// TIA Portal V20 export
FUNCTION_BLOCK "FB_Pos16"   // FB30141, LAD
{ S7_Optimized_Access := 'TRUE' }
// stored: AutoNumber false, MemoryReserve 100, SetENOAutomatically false
   VAR_INPUT
      Opmode { ExternalAccessible := 'False'; ExternalVisible := 'False'; ExternalWritable := 'False'} : "OPMODE_OUT_UDT";
      TO_PosAxis : TO_PositioningAxis;
      I_iNum_Abspos : Int;
      I_bMan_Enable : Bool;
   END_VAR
   VAR_IN_OUT
      Ds_Pos16 : "sPos16";
   END_VAR
   VAR
      instAxis01 { ExternalAccessible := 'False'; ExternalVisible := 'False'; ExternalWritable := 'False'} : "LAxisCtrl_PosAxis";
      instShearAxisStatus { S7_SetPoint := 'True'} : "LAxisCtrl_GetAxisStatusWord";
      RT_Reset { S7_SetPoint := 'True'} : R_TRIG;
      RT_PB { ExternalAccessible := 'False'; ExternalVisible := 'False'; ExternalWritable := 'False'} : Array[0..19] of R_TRIG;   // Störungen / Alarms
      FT_PB { ExternalAccessible := 'False'; ExternalVisible := 'False'; ExternalWritable := 'False'; S7_SetPoint := 'True'} : Array[0..19] of F_TRIG;   // Störungen unterdrücken, Belegung identisch mit "Alarm" / Hide Alarms, identical with "Alarm"
      TON_PB { ExternalAccessible := 'False'; ExternalVisible := 'False'; ExternalWritable := 'False'} : Array[0..19] of TON_TIME;   // Fallende Flanke / Falling edge
      TOF_PB { ExternalAccessible := 'False'; ExternalVisible := 'False'; ExternalWritable := 'False'} : Array[0..19] of TOF_TIME;   // Negativer Impuls / Negative pulse
      i { S7_SetPoint := 'True'} : Int;
      temp_cmd_bEnableAxis { ExternalAccessible := 'False'; ExternalVisible := 'False'; ExternalWritable := 'False'} : Bool;
      temp_cmd_bresetAxis { ExternalAccessible := 'False'; ExternalVisible := 'False'; ExternalWritable := 'False'} : Bool;
      temp_cmd_bjogForward { ExternalAccessible := 'False'; ExternalVisible := 'False'; ExternalWritable := 'False'} : Bool;
      temp_cmd_bjogBackward { ExternalAccessible := 'False'; ExternalVisible := 'False'; ExternalWritable := 'False'} : Bool;
      temp_cmd_bmoveVelocity { ExternalAccessible := 'False'; ExternalVisible := 'False'; ExternalWritable := 'False'} : Bool;
      temp_cmd_bstop { ExternalAccessible := 'False'; ExternalVisible := 'False'; ExternalWritable := 'False'} : Bool;
      temp_cmd_bfastStop { ExternalAccessible := 'False'; ExternalVisible := 'False'; ExternalWritable := 'False'} : Bool;
      temp_cmd_bhoming { ExternalAccessible := 'False'; ExternalVisible := 'False'; ExternalWritable := 'False'} : Bool;
      temp_cmd_bGoToPos { ExternalAccessible := 'False'; ExternalVisible := 'False'; ExternalWritable := 'False'} : Array[0..16] of Bool;
      temp_cmd_iGoToPos : Word;
      temp_cmd_bCallAbsPos : Bool;
      temp_cmd_bRelPos : Bool;
      temp_Para_rJog_Speed { ExternalAccessible := 'False'; ExternalVisible := 'False'; ExternalWritable := 'False'} : LReal;
      temp_configuration { ExternalAccessible := 'False'; ExternalVisible := 'False'; ExternalWritable := 'False'} : "LAxisCtrl_typeAxisConfig";   // Diagnostics structure
      temp_Status { ExternalAccessible := 'False'; ExternalVisible := 'False'; ExternalWritable := 'False'} : Word;
      temp_AxisEnabled { ExternalAccessible := 'False'; ExternalVisible := 'False'; ExternalWritable := 'False'} : Bool;
      temp_CommandBusy { ExternalAccessible := 'False'; ExternalVisible := 'False'; ExternalWritable := 'False'} : Bool;
      temp_CommandDone { ExternalAccessible := 'False'; ExternalVisible := 'False'; ExternalWritable := 'False'} : Bool;
      temp_CommandAborted { ExternalAccessible := 'False'; ExternalVisible := 'False'; ExternalWritable := 'False'} : Bool;
      temp_InVelocity { ExternalAccessible := 'False'; ExternalVisible := 'False'; ExternalWritable := 'False'} : Bool;
      temp_jogSelected { ExternalAccessible := 'False'; ExternalVisible := 'False'; ExternalWritable := 'False'} : Bool;
      tempPosAbsoluteSelected { ExternalAccessible := 'False'; ExternalVisible := 'False'; ExternalWritable := 'False'} : Bool;
      temp_diagnostics { ExternalAccessible := 'False'; ExternalVisible := 'False'; ExternalWritable := 'False'} : "LAxisCtrl_typeDiagnostics";
      temp_stop_Dec { ExternalAccessible := 'False'; ExternalVisible := 'False'; ExternalWritable := 'False'} : LReal;
      temp_faststop_Dec { ExternalAccessible := 'False'; ExternalVisible := 'False'; ExternalWritable := 'False'} : LReal;
      temp_cmd_bGoToPosAll : Bool;
      temp_iFBStatus : Word;
      temp_iMCStatus : Word;
      old_iFBStatus : Word;
      old_iMCStatus : Word;
   END_VAR
BEGIN

REGION Network 1
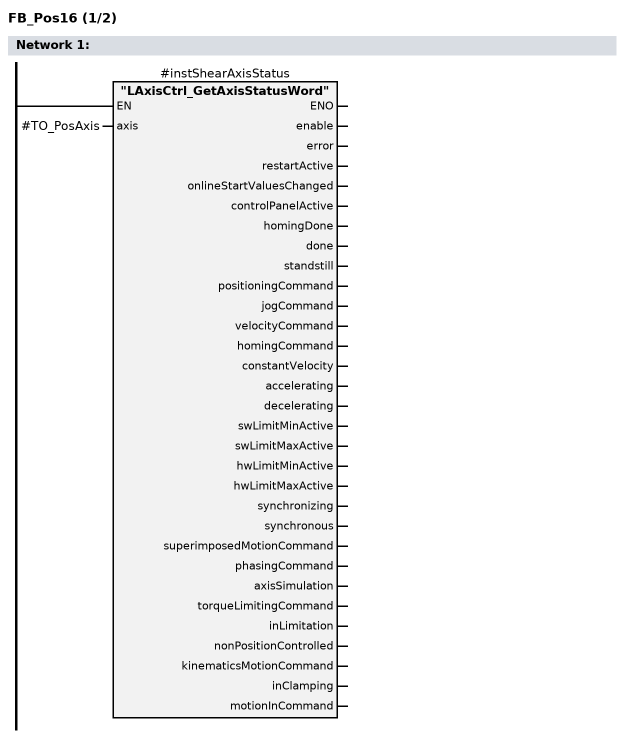
   RUNG wire#powerrail
      #instShearAxisStatus(axis := #TO_PosAxis, enable =>, error =>, restartActive =>, onlineStartValuesChanged =>, controlPanelActive =>, homingDone =>, done =>, standstill =>, positioningCommand =>, jogCommand =>, velocityCommand =>, homingCommand =>, constantVelocity =>, accelerating =>, decelerating =>, swLimitMinActive =>, swLimitMaxActive =>, hwLimitMinActive =>, hwLimitMaxActive =>, synchronizing =>, synchronous =>, superimposedMotionCommand =>, phasingCommand =>, axisSimulation =>, torqueLimitingCommand =>, inLimitation =>, nonPositionControlled =>, kinematicsMotionCommand =>, inClamping =>, motionInCommand =>)
   END_RUNG
   // the same network as SCL:
   #instShearAxisStatus(axis := #TO_PosAxis);   // "LAxisCtrl_GetAxisStatusWord"
END_REGION

REGION Network 2: LAxisCtrl
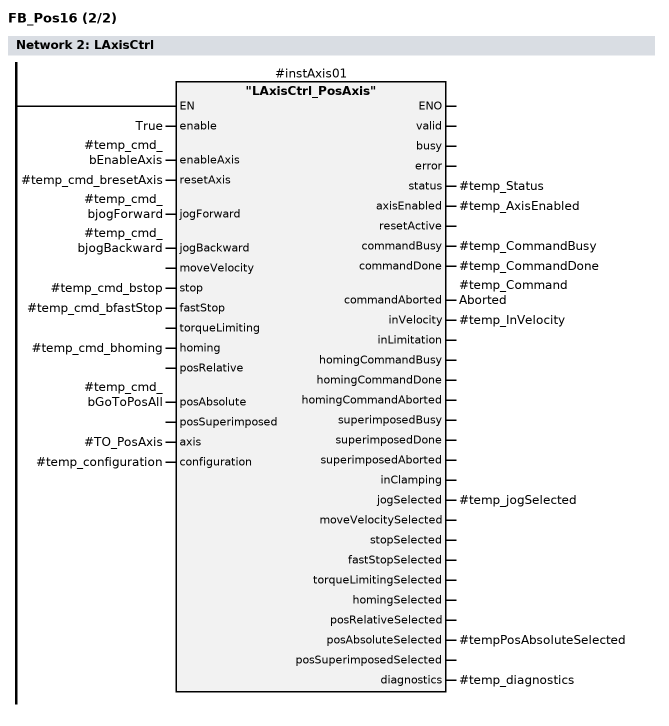
   RUNG wire#powerrail
      #instAxis01(enable := True, enableAxis := #temp_cmd_bEnableAxis, resetAxis := #temp_cmd_bresetAxis, jogForward := #temp_cmd_bjogForward, jogBackward := #temp_cmd_bjogBackward, moveVelocity :=, stop := #temp_cmd_bstop, fastStop := #temp_cmd_bfastStop, torqueLimiting :=, homing := #temp_cmd_bhoming, posRelative :=, posAbsolute := #temp_cmd_bGoToPosAll, posSuperimposed :=, axis := #TO_PosAxis, configuration := #temp_configuration, valid =>, busy =>, error =>, status => #temp_Status, axisEnabled => #temp_AxisEnabled, resetActive =>, commandBusy => #temp_CommandBusy, commandDone => #temp_CommandDone, commandAborted => #temp_CommandAborted, inVelocity => #temp_InVelocity, inLimitation =>, homingCommandBusy =>, homingCommandDone =>, homingCommandAborted =>, superimposedBusy =>, superimposedDone =>, superimposedAborted =>, inClamping =>, jogSelected => #temp_jogSelected, moveVelocitySelected =>, stopSelected =>, fastStopSelected =>, torqueLimitingSelected =>, homingSelected =>, posRelativeSelected =>, posAbsoluteSelected => #tempPosAbsoluteSelected, posSuperimposedSelected =>, diagnostics => #temp_diagnostics)
   END_RUNG
   // the same network as SCL:
   #instAxis01(enable := True,   // "LAxisCtrl_PosAxis"
               enableAxis := #temp_cmd_bEnableAxis,
               resetAxis := #temp_cmd_bresetAxis,
               jogForward := #temp_cmd_bjogForward,
               jogBackward := #temp_cmd_bjogBackward,
               stop := #temp_cmd_bstop,
               fastStop := #temp_cmd_bfastStop,
               homing := #temp_cmd_bhoming,
               posAbsolute := #temp_cmd_bGoToPosAll,
               axis := #TO_PosAxis,
               configuration := #temp_configuration,
               status => #temp_Status,
               axisEnabled => #temp_AxisEnabled,
               commandBusy => #temp_CommandBusy,
               commandDone => #temp_CommandDone,
               commandAborted => #temp_CommandAborted,
               inVelocity => #temp_InVelocity,
               jogSelected => #temp_jogSelected,
               posAbsoluteSelected => #tempPosAbsoluteSelected,
               diagnostics => #temp_diagnostics);
END_REGION

REGION Network 3 (SCL): input
   #temp_cmd_bEnableAxis  := #Ds_Pos16.I_CMD_bEnableAxis OR (#Ds_Pos16.I_HMI_bEnableAxis AND #I_bMan_Enable);
   #temp_cmd_bresetAxis   := #Ds_Pos16.I_CMD_bResetAxis;
   #temp_cmd_bjogForward  := #Ds_Pos16.I_InLock_bjogForward AND (#Ds_Pos16.I_CMD_bjogForward OR (#Ds_Pos16.I_HMI_bjogForward AND #I_bMan_Enable));
   #temp_cmd_bjogBackward := #Ds_Pos16.I_InLock_bjogBackward AND (#Ds_Pos16.I_CMD_bjogBackward OR (#Ds_Pos16.I_HMI_bjogBackward AND #I_bMan_Enable));
   #temp_cmd_bstop        := #Ds_Pos16.I_CMD_bstop OR (#Ds_Pos16.I_HMI_bstop AND #I_bMan_Enable);
   #temp_cmd_bfastStop    := #Ds_Pos16.I_CMD_bfastStop;
   #temp_cmd_bhoming      := #Ds_Pos16.I_InLock_bHoming AND (#Ds_Pos16.I_CMD_bHoming OR #Ds_Pos16.I_HMI_bHoming);
END_REGION

REGION Network 4 (SCL): Configuration
   #Ds_Pos16.I_Para_rJog_Speed[0] := 10.0;
   #Ds_Pos16.I_Para_rMV_Speed[0]  := 10.0;
   #Ds_Pos16.I_Para_rStop_Dec[0]  := 20.0;
   #Ds_Pos16.I_Para_rEStop_Dec[0] := 50.0;

   #Ds_Pos16.I_Para_rJog_Speed[1] := 10.0 * #Ds_Pos16.I_Para_rJog_Speed[0];
   #Ds_Pos16.I_Para_rJog_Speed[2] := 10.0 * #Ds_Pos16.I_Para_rJog_Speed[0];
   #Ds_Pos16.I_Para_rMV_Speed[1] := 10.0 * #Ds_Pos16.I_Para_rMV_Speed[0];
   #Ds_Pos16.I_Para_rMV_Speed[2] := 10.0 * #Ds_Pos16.I_Para_rMV_Speed[0];
   #Ds_Pos16.I_Para_rStop_Dec[1] := 100.0 * #Ds_Pos16.I_Para_rStop_Dec[0];
   #Ds_Pos16.I_Para_rEStop_Dec[1] := 100.0 * #Ds_Pos16.I_Para_rEStop_Dec[0];

   IF #temp_configuration.jog.velocity <> #Ds_Pos16.I_Para_rJog_Speed[0] OR
       #temp_configuration.jog.acceleration <> #Ds_Pos16.I_Para_rJog_Speed[1] OR
       #temp_configuration.jog.deceleration <> #Ds_Pos16.I_Para_rJog_Speed[2] OR
       #temp_configuration.moveVelocity.acceleration <> #Ds_Pos16.I_Para_rMV_Speed[0] OR
       #temp_configuration.moveVelocity.deceleration <> #Ds_Pos16.I_Para_rMV_Speed[1] OR
       #temp_configuration.moveVelocity.acceleration <> #Ds_Pos16.I_Para_rMV_Speed[2] OR
       #temp_configuration.stop.deceleration <> #Ds_Pos16.I_Para_rStop_Dec[0] OR
       #temp_configuration.stop.jerk <> #Ds_Pos16.I_Para_rStop_Dec[1] OR
       #temp_configuration.fastStop.deceleration <> #Ds_Pos16.I_Para_rEStop_Dec[0] OR
       #temp_configuration.fastStop.jerk <> #Ds_Pos16.I_Para_rEStop_Dec[1]
   THEN
       // Jog
       #temp_configuration.jog.velocity := #Ds_Pos16.I_Para_rJog_Speed[0];
       #temp_configuration.jog.acceleration := #Ds_Pos16.I_Para_rJog_Speed[1];
       #temp_configuration.jog.deceleration := #Ds_Pos16.I_Para_rJog_Speed[2];
       // Move
       #temp_configuration.moveVelocity.velocity := #Ds_Pos16.I_Para_rMV_Speed[0];
       #temp_configuration.moveVelocity.acceleration := #Ds_Pos16.I_Para_rMV_Speed[1];
       #temp_configuration.moveVelocity.deceleration := #Ds_Pos16.I_Para_rMV_Speed[2];
       // Stop   
       #temp_configuration.stop.deceleration := #Ds_Pos16.I_Para_rStop_Dec[0];
       #temp_configuration.stop.jerk := #Ds_Pos16.I_Para_rStop_Dec[1];
       //faststoo
       #temp_configuration.fastStop.deceleration := #Ds_Pos16.I_Para_rEStop_Dec[0];
       #temp_configuration.fastStop.jerk := #Ds_Pos16.I_Para_rEStop_Dec[1];
   END_IF;

   // Homing
   #temp_configuration.homing.mode := 0;//I_iHomeMode
   #temp_configuration.homing.position := 0;//I_iHomePos

   //abspos
   FOR #i := 1 TO 16 DO
       #Ds_Pos16.I_Para_rAcc_Set[#i] := 10.0 * #Ds_Pos16.I_Para_rSpeed_Abs[0];
       #Ds_Pos16.I_Para_rDec_Set[#i] := 10.0 * #Ds_Pos16.I_Para_rSpeed_Abs[0];
       #Ds_Pos16.I_Para_rJerk_Set[#i] := 100.0 * #Ds_Pos16.I_Para_rSpeed_Abs[0];
   END_FOR;


   //#temp_posAbsolute := (#Ds_Pos16.I_CMD_iGoToPos <> 16#0);
   #temp_cmd_bGoToPos[1] := ((#Opmode.Automatic_active=1 AND #Ds_Pos16.I_CMD_iGoToPos = 1) OR (#Opmode.Manual_active AND #Ds_Pos16.I_HMI_iGoToPos = 1)) AND #Ds_Pos16.I_InLock_bGoToPos[1];
   #temp_cmd_bGoToPos[2] := ((#Opmode.Automatic_active=1 AND #Ds_Pos16.I_CMD_iGoToPos = 2) OR (#Opmode.Manual_active AND  #Ds_Pos16.I_HMI_iGoToPos = 2)) AND #Ds_Pos16.I_InLock_bGoToPos[2];
   #temp_cmd_bGoToPos[3] := ((#Opmode.Automatic_active=1 AND #Ds_Pos16.I_CMD_iGoToPos = 3) OR (#Opmode.Manual_active AND  #Ds_Pos16.I_HMI_iGoToPos = 3)) AND #Ds_Pos16.I_InLock_bGoToPos[3];
   #temp_cmd_bGoToPos[4] := ((#Opmode.Automatic_active=1 AND #Ds_Pos16.I_CMD_iGoToPos = 4) OR (#Opmode.Manual_active AND  #Ds_Pos16.I_HMI_iGoToPos = 4)) AND #Ds_Pos16.I_InLock_bGoToPos[4];
   #temp_cmd_bGoToPos[5] := ((#Opmode.Automatic_active=1 AND #Ds_Pos16.I_CMD_iGoToPos = 5) OR (#Opmode.Manual_active AND  #Ds_Pos16.I_HMI_iGoToPos = 5)) AND #Ds_Pos16.I_InLock_bGoToPos[5];
   #temp_cmd_bGoToPos[6] := ((#Opmode.Automatic_active=1 AND #Ds_Pos16.I_CMD_iGoToPos = 6) OR (#Opmode.Manual_active AND  #Ds_Pos16.I_HMI_iGoToPos = 6)) AND #Ds_Pos16.I_InLock_bGoToPos[6];
   #temp_cmd_bGoToPos[7] := ((#Opmode.Automatic_active=1 AND #Ds_Pos16.I_CMD_iGoToPos = 7) OR (#Opmode.Manual_active AND  #Ds_Pos16.I_HMI_iGoToPos = 7)) AND #Ds_Pos16.I_InLock_bGoToPos[7];
   #temp_cmd_bGoToPos[8] := ((#Opmode.Automatic_active=1 AND #Ds_Pos16.I_CMD_iGoToPos = 8) OR (#Opmode.Manual_active AND  #Ds_Pos16.I_HMI_iGoToPos = 8)) AND #Ds_Pos16.I_InLock_bGoToPos[8];
   #temp_cmd_bGoToPos[9] := ((#Opmode.Automatic_active=1 AND #Ds_Pos16.I_CMD_iGoToPos = 9) OR (#Opmode.Manual_active AND  #Ds_Pos16.I_HMI_iGoToPos = 9)) AND #Ds_Pos16.I_InLock_bGoToPos[9];
   #temp_cmd_bGoToPos[10] := ((#Opmode.Automatic_active=1 AND #Ds_Pos16.I_CMD_iGoToPos = 10) OR (#Opmode.Manual_active AND  #Ds_Pos16.I_HMI_iGoToPos = 10)) AND #Ds_Pos16.I_InLock_bGoToPos[10];
   #temp_cmd_bGoToPos[11] := ((#Opmode.Automatic_active=1 AND #Ds_Pos16.I_CMD_iGoToPos = 11) OR (#Opmode.Manual_active AND  #Ds_Pos16.I_HMI_iGoToPos = 11)) AND #Ds_Pos16.I_InLock_bGoToPos[11];
   #temp_cmd_bGoToPos[12] := ((#Opmode.Automatic_active=1 AND #Ds_Pos16.I_CMD_iGoToPos = 12) OR (#Opmode.Manual_active AND  #Ds_Pos16.I_HMI_iGoToPos = 12)) AND #Ds_Pos16.I_InLock_bGoToPos[12];
   #temp_cmd_bGoToPos[13] := ((#Opmode.Automatic_active=1 AND #Ds_Pos16.I_CMD_iGoToPos = 13) OR (#Opmode.Manual_active AND  #Ds_Pos16.I_HMI_iGoToPos = 13)) AND #Ds_Pos16.I_InLock_bGoToPos[13];
   #temp_cmd_bGoToPos[14] := ((#Opmode.Automatic_active=1 AND #Ds_Pos16.I_CMD_iGoToPos = 14) OR (#Opmode.Manual_active AND  #Ds_Pos16.I_HMI_iGoToPos = 14)) AND #Ds_Pos16.I_InLock_bGoToPos[14];
   #temp_cmd_bGoToPos[15] := ((#Opmode.Automatic_active=1 AND #Ds_Pos16.I_CMD_iGoToPos = 15) OR (#Opmode.Manual_active AND  #Ds_Pos16.I_HMI_iGoToPos = 15)) AND #Ds_Pos16.I_InLock_bGoToPos[15];
   #temp_cmd_bGoToPos[16] := ((#Opmode.Automatic_active=1 AND #Ds_Pos16.I_CMD_iGoToPos = 16) OR (#Opmode.Manual_active AND  #Ds_Pos16.I_HMI_iGoToPos = 16)) AND #Ds_Pos16.I_InLock_bGoToPos[16];

   #temp_cmd_bGoToPosAll := #temp_cmd_bGoToPos[1] OR #temp_cmd_bGoToPos[2] OR #temp_cmd_bGoToPos[3] OR #temp_cmd_bGoToPos[4]
   OR #temp_cmd_bGoToPos[5] OR #temp_cmd_bGoToPos[6] OR #temp_cmd_bGoToPos[7] OR #temp_cmd_bGoToPos[8]
   OR #temp_cmd_bGoToPos[9] OR #temp_cmd_bGoToPos[10] OR #temp_cmd_bGoToPos[11] OR #temp_cmd_bGoToPos[12]
   OR #temp_cmd_bGoToPos[13] OR #temp_cmd_bGoToPos[14] OR #temp_cmd_bGoToPos[15] OR #temp_cmd_bGoToPos[16]
   ;
   //#temp_posAbsolute :=
   //#Ds_Pos16.I_bGoToPos[0] OR #Ds_Pos16.I_bGoToPos[1] OR #Ds_Pos16.I_bGoToPos[2] OR #Ds_Pos16.I_bGoToPos[3] OR
   //#Ds_Pos16.I_bGoToPos[4] OR #Ds_Pos16.I_bGoToPos[5] OR #Ds_Pos16.I_bGoToPos[6] OR #Ds_Pos16.I_bGoToPos[7] OR
   //#Ds_Pos16.I_bGoToPos[8] OR #Ds_Pos16.I_bGoToPos[9] OR #Ds_Pos16.I_bGoToPos[10] OR #Ds_Pos16.I_bGoToPos[11] OR
   //#Ds_Pos16.I_bGoToPos[12] OR #Ds_Pos16.I_bGoToPos[13] OR #Ds_Pos16.I_bGoToPos[14] OR #Ds_Pos16.I_bGoToPos[15];

   FOR #i := 1 TO 16 DO
   //    #RT_PB[#i](CLK := #Ds_Pos16.I_bGoToPos[#i]);
       #RT_PB[#i](CLK := #temp_cmd_bGoToPos[#i]);

       IF #RT_PB[#i].Q THEN
           #temp_configuration.posAbsolute.position := #Ds_Pos16.I_Para_rPos_Abs[#i];
           #temp_configuration.posAbsolute.velocity := #Ds_Pos16.I_Para_rSpeed_Abs[#i];
           #temp_configuration.posAbsolute.direction := 3;//temp_posAbsolute_direction

           #temp_configuration.posAbsolute.acceleration := #Ds_Pos16.I_Para_rAcc_Set[#i];
           #temp_configuration.posAbsolute.deceleration := #Ds_Pos16.I_Para_rDec_Set[#i];
           #temp_configuration.posAbsolute.jerk := #Ds_Pos16.I_Para_rJerk_Set[#i];

       END_IF;
   END_FOR;
END_REGION

REGION Network 5 (SCL): output
   #Ds_Pos16.O_Status_bAxisReady := true;//#TO_PosAxis.StatusWord.%X1;
   #Ds_Pos16.O_Status_bAxisEnabled := #temp_AxisEnabled;
   #Ds_Pos16.O_Status_bjogForward := #temp_cmd_bjogForward;// AND #temp_jogSelected;
   #Ds_Pos16.O_Status_bjogBackward := #temp_cmd_bjogBackward;// AND #temp_jogSelected;
   #Ds_Pos16.O_Status_bHomed := #TO_PosAxis.StatusWord.%X5;
   #Ds_Pos16.O_Status_bAxisError := #TO_PosAxis.StatusWord.%X1;
   #Ds_Pos16.O_Status_rActPos := #TO_PosAxis.ActualPosition;
   #Ds_Pos16.O_Status_rActSpeed := #TO_PosAxis.ActualVelocity;
   #Ds_Pos16.O_Status_iAxisFaultNum := #TO_PosAxis.ErrorDetail.Number;
   //#Ds_Pos16.O_DriveFaultNum
   //#Ds_Pos16.O_Status_iFBStatus := #temp_diagnostics.status;
   //#Ds_Pos16.O_Status_iMCStatus := #temp_diagnostics.subfunctionStatus;
   //#Ds_Pos16.O_Torque
   //#Ds_Pos16.oAxisName  := 

   FOR #i := 0 TO 15 DO
       #Ds_Pos16.O_Status_bAtPos[#i] := "FC_bNearIn"(rAct := #Ds_Pos16.O_Status_rActPos, rTgt := #Ds_Pos16.I_Para_rPos_Abs[#i], rDelta := 1.0, bModule := 0, rModulo := 0);
   END_FOR;

   //#Ds_Pos16.O_bPosDone
   //#Ds_Pos16.O_bPosing
   //#tempPosAbsoluteSelected
END_REGION

REGION Network 6 (SCL): Reset
   #RT_Reset(CLK := #temp_cmd_bresetAxis);
   IF #RT_Reset.Q THEN
       #Ds_Pos16.O_Status_iFBStatus := 16#00;
       #Ds_Pos16.O_Status_iMCStatus := 16#00;
   END_IF;

   #temp_iFBStatus := #temp_diagnostics.status;
   IF #temp_iFBStatus <> #old_iFBStatus THEN
       #Ds_Pos16.O_Status_iFBStatus := #temp_diagnostics.status;
       #old_iFBStatus := #temp_iFBStatus;
   END_IF;
   #temp_iMCStatus := #temp_diagnostics.subfunctionStatus;
   IF #temp_iMCStatus <> #old_iMCStatus THEN
       #Ds_Pos16.O_Status_iFBStatus := #temp_diagnostics.subfunctionStatus;
       #old_iMCStatus := #temp_iMCStatus;
   END_IF;
END_REGION

REGION Network 7 (SCL)
   (*
   FOR #i := 9 TO 16 DO
       IF #I_iNum_Abspos < #i THEN
           #Ds_Pos16.I_InLock_bGoToPos[#i] := false;
       END_IF;
   END_FOR;
   *)
END_REGION
END_FUNCTION_BLOCK
